// TIA Portal project "sorting_station" (V15.1)
// Vorlageprojekt für das Buch mit Zielsystem S7-1200

(* hardware
DEVICE "S7-1200-Station_1"  S7-1200 Station
   slot 0: "Baugruppenträger_0"  Rack  V1.0
   slot 1: "PLC_1"  CPU 1211C DC/DC/DC  6ES7 211-1AE40-0XB0  V4.1
*)

// ===== PLC "PLC_1"  CPU 1211C DC/DC/DC =====

VAR_GLOBAL   // PLC tag table "Standard-Variablentabelle"
   "Entry Conveyor" AT %A0.0 : Bool;
   "Start" AT %E0.1 : Bool;
   "Stop" AT %I0.3 : Bool;
   "Vision Sensor" AT %ID30 : DWord;
   "Green Sorter Turn" AT %Q0.3 : Bool;
   "Blue Sorter Turn" AT %Q0.7 : Bool;
   "Exit Conveyor" AT %Q0.2 : Bool;
   "Gray Sorter Turn" AT %Q0.5 : Bool;
   "Gray Timer Valve" AT %Q1.4 : Bool;
   "Green Sorter Belt" AT %Q0.4 : Bool;
   "Gray Sorter Belt" AT %Q0.6 : Bool;
   "Blue Sorter Belt" AT %Q1.0 : Bool;
   "Green Timer Valve" AT %Q1.5 : Bool;
   "Blue Timer Valve" AT %Q1.6 : Bool;
   "Counter 1" AT %QD30 : DWord;
   "Reset" AT %I0.2 : Bool;
   "Counter 2" AT %QD34 : DWord;
   "Counter 3" AT %QD38 : DWord;
END_VAR

// folder: System blocks/Program resources

DATA_BLOCK "IEC_Timer_0_DB"   // DB1
{ S7_Optimized_Access := 'TRUE' }
AUTHOR : Simatic
FAMILY : IEC
NAME : IEC_TMR
VERSION : 1.0
// stored: InstanceOfName IEC_TIMER
"IEC_TIMER"
BEGIN
END_DATA_BLOCK

DATA_BLOCK "IEC_Timer_0_DB_1"   // DB2
{ S7_Optimized_Access := 'TRUE' }
AUTHOR : Simatic
FAMILY : IEC
NAME : IEC_TMR
VERSION : 1.0
// stored: InstanceOfName IEC_TIMER
"IEC_TIMER"
BEGIN
END_DATA_BLOCK

DATA_BLOCK "IEC_Timer_0_DB_2"   // DB3
{ S7_Optimized_Access := 'TRUE' }
AUTHOR : Simatic
FAMILY : IEC
NAME : IEC_TMR
VERSION : 1.0
// stored: InstanceOfName IEC_TIMER
"IEC_TIMER"
BEGIN
END_DATA_BLOCK

DATA_BLOCK "IEC_Timer_0_DB_3"   // DB4
{ S7_Optimized_Access := 'TRUE' }
AUTHOR : Simatic
FAMILY : IEC
NAME : IEC_TMR
VERSION : 1.0
// stored: InstanceOfName IEC_TIMER
"IEC_TIMER"
BEGIN
END_DATA_BLOCK

DATA_BLOCK "IEC_Timer_0_DB_4"   // DB5
{ S7_Optimized_Access := 'TRUE' }
AUTHOR : Simatic
FAMILY : IEC
NAME : IEC_TMR
VERSION : 1.0
// stored: InstanceOfName IEC_TIMER
"IEC_TIMER"
BEGIN
END_DATA_BLOCK

DATA_BLOCK "IEC_Timer_0_DB_5"   // DB6
{ S7_Optimized_Access := 'TRUE' }
AUTHOR : Simatic
FAMILY : IEC
NAME : IEC_TMR
VERSION : 1.0
// stored: InstanceOfName IEC_TIMER
"IEC_TIMER"
BEGIN
END_DATA_BLOCK

DATA_BLOCK "IEC_Counter_0_DB"   // DB7
{ S7_Optimized_Access := 'TRUE' }
AUTHOR : Simatic
FAMILY : IEC
NAME : CNTR
VERSION : 1.0
// stored: InstanceOfName IEC_COUNTER
"IEC_COUNTER"
BEGIN
END_DATA_BLOCK

DATA_BLOCK "IEC_Counter_0_DB_1"   // DB8
{ S7_Optimized_Access := 'TRUE' }
AUTHOR : Simatic
FAMILY : IEC
NAME : CNTR
VERSION : 1.0
// stored: InstanceOfName IEC_COUNTER
"IEC_COUNTER"
BEGIN
END_DATA_BLOCK

DATA_BLOCK "IEC_Counter_0_DB_2"   // DB9
{ S7_Optimized_Access := 'TRUE' }
AUTHOR : Simatic
FAMILY : IEC
NAME : CNTR
VERSION : 1.0
// stored: InstanceOfName IEC_COUNTER
"IEC_COUNTER"
BEGIN
END_DATA_BLOCK

// folder: (top level)

FUNCTION "MHJ-PLC-Lab-Function-S71200" : Void   // FC9000, SCL
{ S7_Optimized_Access := 'TRUE' }
VERSION : 0.1
   VAR_TEMP
      rdTimeReturn : Int;
      outputTime : DTL;
      SyncVal : Byte;
      forVal : Int;
      forVal_2 : Int;
      Value : Byte;
   END_VAR
   VAR CONSTANT
      CompVal : Byte := 16#34;
      Value_01 : Byte := 16#11;
      Value_01_DW : DWord := 16#A165_D992;
      Value_02_DW : DWord := 16#58BE_4401;
   END_VAR
BEGIN

   #Value:=PEEK(area := 16#82,
        dbNumber := 0,
        byteOffset := 511);
   #Value := #Value + 1;

   POKE(area := 16#82,
        dbNumber := 0,
        byteOffset := 511,
        value := #Value);

   POKE(area:=16#81,
        dbNumber:=0,
        byteOffset:=1016,
        value:=#Value_01_DW);
   POKE(area := 16#81,
        dbNumber := 0,
        byteOffset := 1020,
        value := #Value_02_DW);

   POKE(area := 16#81,
        dbNumber := 0,
        byteOffset := 511,
        value := B#16#00);

   FOR #forVal := 0 TO 120 DO
       FOR #forVal_2:=0 TO 10 DO
           #rdTimeReturn:=RD_SYS_T(#outputTime);
           #rdTimeReturn := WR_SYS_T(#outputTime);
           #rdTimeReturn := RD_SYS_T(#outputTime);
           #rdTimeReturn := WR_SYS_T(#outputTime);
       END_FOR;
       #SyncVal:= PEEK(area := 16#81,
                      dbNumber := 0,
                      byteOffset := 511);
       IF #SyncVal = #CompVal THEN
          GOTO M_1;
       END_IF;
   END_FOR;
   RETURN;

   M_1:
   POKE(area := 16#81,
        dbNumber := 0,
        byteOffset := 511,
        value := B#16#0);
END_FUNCTION

ORGANIZATION_BLOCK "Main"   // OB1, LAD, ProgramCycle
TITLE = "Main Program Sweep (Cycle)"
{ S7_Optimized_Access := 'TRUE' }
VERSION : 0.1
   VAR_INPUT
      Initial_Call : Bool;   // Initial call of this OB
      Remanence : Bool;   // =True, if remanent data are available
   END_VAR
BEGIN

REGION Network 1: Konnektierungsbaustein für PLC-Lab
   // Im Netzwerk 1 wird der Konnektierungsbaustein für PLC-Lab aufgerufen.
   // Dieser Aufruf darf nicht entfernt werden!
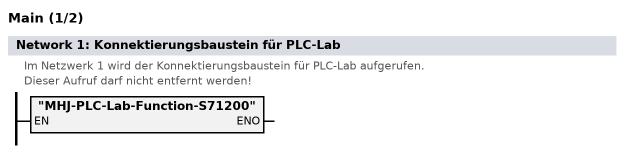
   RUNG wire#powerrail
      "MHJ-PLC-Lab-Function-S71200"()
   END_RUNG
   // the same network as SCL:
   "MHJ-PLC-Lab-Function-S71200"();
END_REGION

REGION Network 2: Ihr Programm
   // Schreiben Sie ab Netzwerk 2 Ihr Programm
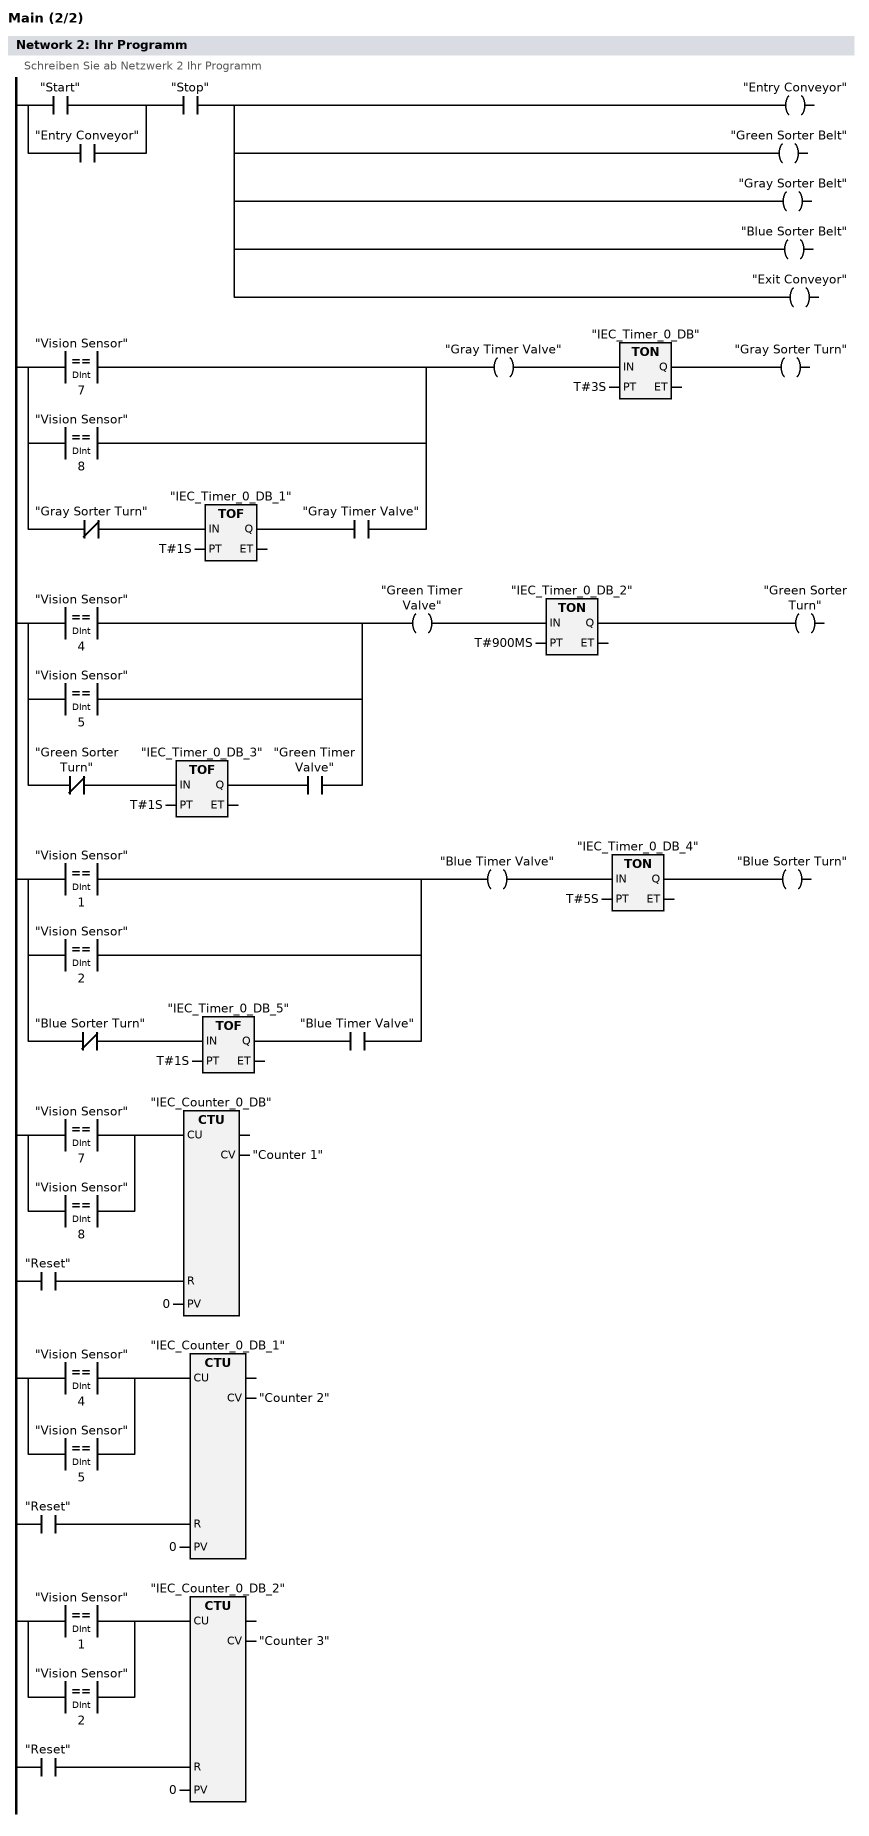
   "Entry Conveyor" := ("Start" OR "Entry Conveyor") AND "Stop";
   "Green Sorter Belt" := "Entry Conveyor";
   "Gray Sorter Belt" := "Entry Conveyor";
   "Blue Sorter Belt" := "Entry Conveyor";
   "Exit Conveyor" := "Entry Conveyor";
   "IEC_Timer_0_DB_1".TOF(IN := NOT "Gray Sorter Turn", PT := T#1S);
   "Gray Timer Valve" := ("Vision Sensor" = 7) OR ("Vision Sensor" = 8) OR ("IEC_Timer_0_DB_1".Q AND "Gray Timer Valve");
   "IEC_Timer_0_DB".TON(IN := "Gray Timer Valve", PT := T#3S);
   "Gray Sorter Turn" := "IEC_Timer_0_DB".Q;
   "IEC_Timer_0_DB_3".TOF(IN := NOT "Green Sorter Turn", PT := T#1S);
   "Green Timer Valve" := ("Vision Sensor" = 4) OR ("Vision Sensor" = 5) OR ("IEC_Timer_0_DB_3".Q AND "Green Timer Valve");
   "IEC_Timer_0_DB_2".TON(IN := "Green Timer Valve", PT := T#900MS);
   "Green Sorter Turn" := "IEC_Timer_0_DB_2".Q;
   "IEC_Timer_0_DB_5".TOF(IN := NOT "Blue Sorter Turn", PT := T#1S);
   "Blue Timer Valve" := ("Vision Sensor" = 1) OR ("Vision Sensor" = 2) OR ("IEC_Timer_0_DB_5".Q AND "Blue Timer Valve");
   "IEC_Timer_0_DB_4".TON(IN := "Blue Timer Valve", PT := T#5S);
   "Blue Sorter Turn" := "IEC_Timer_0_DB_4".Q;
   "IEC_Counter_0_DB".CTU(CU := ("Vision Sensor" = 7) OR ("Vision Sensor" = 8),
                          R := "Reset",
                          PV := 0,
                          CV => "Counter 1");
   "IEC_Counter_0_DB_1".CTU(CU := ("Vision Sensor" = 4) OR ("Vision Sensor" = 5),
                           R := "Reset",
                           PV := 0,
                           CV => "Counter 2");
   "IEC_Counter_0_DB_2".CTU(CU := ("Vision Sensor" = 1) OR ("Vision Sensor" = 2),
                           R := "Reset",
                           PV := 0,
                           CV => "Counter 3");
END_REGION
END_ORGANIZATION_BLOCK